// TIA Portal V19 export
FUNCTION "A0301_Fermi_P3_CALL" : Void   // FC120, LAD
// stored: SetENOAutomatically false
BEGIN

REGION Network 1 (SCL): << TRASFERIMENTO stati CIn del blocco >>
   // TRASFERIMENTO #CIn MANAGER
   "A0301_Fermi_P3".CIn.Manager := "A0301_Manager".COut.P3.Fermi;
   //
   "A0301_Fermi_P3".CIn.SemiAut := "A0301_Manager".DataIn.SemiAut_Pb;

   // Trasferimento status alla Stazione P2 da COut a Cin delle stazioni successive
   "A0301_Fermi_P3".CIn.P2.Fermi := "A0301_Fermi_P2".COut.Fermi;

   // Trasferimento status alla Stazione P3 da COut a Cin del sollevatore P2
   "A0301_Fermi_P3".CIn.P2.Sollevatore := "A0301_Fermi_P2".COut.Sollevatori;

   // Trasferimenti status lettura posizioni Trasporto al Cin delle stazioni
   "A0301_Fermi_P3".CIn.Trasporto := "A0301_Trasporto".COut.Ax;
END_REGION

REGION Network 2 (SCL): << TRASFERIMENTO stati DataIn >>
   // SOSTITUIRE SYS.BAYPASS
   // TRASFERIMENTO #DataIn STATI BUTTON STAZIONE P3

   REGION TRASFERIMENTO DataIn DIGITAL INPUT dei LIMIT SWITCH

       // Trasferimento ingressi digitali Limit Switch Fermi P3
       // 
       "A0301_Fermi_P3".Fermi[1].DataIn.Rest_Ls[1] := "A0301_CinghiaTrasporto_1.2_Ls_Rest_1";
       "A0301_Fermi_P3".Fermi[2].DataIn.Rest_Ls[1] := "A0301_CinghiaTrasporto_2.2_Ls_Rest_1";
       "A0301_Fermi_P3".Fermi[3].DataIn.Rest_Ls[1] := "A0301_CinghiaTrasporto_3.2_Ls_Rest_1";
       "A0301_Fermi_P3".Fermi[4].DataIn.Rest_Ls[1] := "A0301_CinghiaTrasporto_4.2_Ls_Rest_1";
       "A0301_Fermi_P3".Fermi[5].DataIn.Rest_Ls[1] := "A0301_CinghiaTrasporto_5.2_Ls_Rest_1";
       "A0301_Fermi_P3".Fermi[6].DataIn.Rest_Ls[1] := "A0301_CinghiaTrasporto_6.2_Ls_Rest_1";

   END_REGION ;
END_REGION

REGION Network 3: DataIn - Fermi
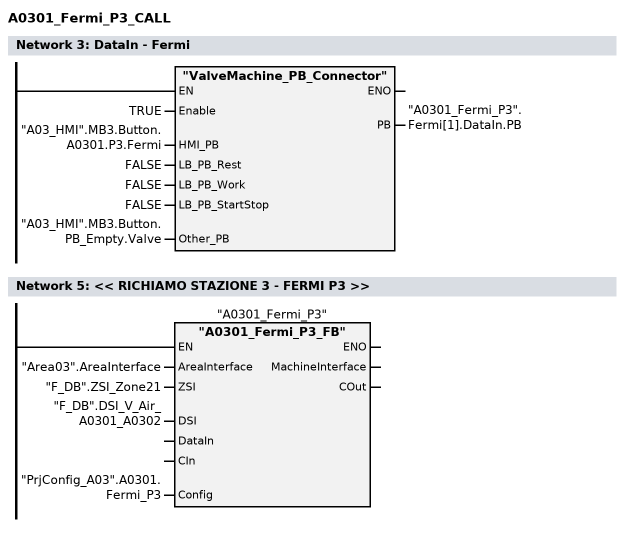
   RUNG wire#powerrail
      "ValveMachine_PB_Connector"(Enable := TRUE, HMI_PB := "A03_HMI".MB3.Button.A0301.P3.Fermi, LB_PB_Rest := FALSE, LB_PB_Work := FALSE, LB_PB_StartStop := FALSE, Other_PB := "A03_HMI".MB3.Button.PB_Empty.Valve, PB => "A0301_Fermi_P3".Fermi[1].DataIn.PB)
   END_RUNG
   // the same network as SCL:
   "ValveMachine_PB_Connector"(Enable := TRUE,
                           HMI_PB := "A03_HMI".MB3.Button.A0301.P3.Fermi,
                           LB_PB_Rest := FALSE,
                           LB_PB_Work := FALSE,
                           LB_PB_StartStop := FALSE,
                           Other_PB := "A03_HMI".MB3.Button.PB_Empty.Valve,
                           PB => "A0301_Fermi_P3".Fermi[1].DataIn.PB);
END_REGION

REGION Network 4 (SCL): DataIn - Fermi [1..6]
   // TRASFERIMENTO STATO PULSANTI - Comando manuale diretto 
   "A0301_Fermi_P3".Fermi[6].DataIn.PB.Rest := "A0301_Fermi_P3".Fermi[5].DataIn.PB.Rest := "A0301_Fermi_P3".Fermi[4].DataIn.PB.Rest :=
   "A0301_Fermi_P3".Fermi[3].DataIn.PB.Rest := "A0301_Fermi_P3".Fermi[2].DataIn.PB.Rest := "A0301_Fermi_P3".Fermi[1].DataIn.PB.Rest;

   "A0301_Fermi_P3".Fermi[6].DataIn.PB.Work := "A0301_Fermi_P3".Fermi[5].DataIn.PB.Work := "A0301_Fermi_P3".Fermi[4].DataIn.PB.Work :=
   "A0301_Fermi_P3".Fermi[3].DataIn.PB.Work := "A0301_Fermi_P3".Fermi[2].DataIn.PB.Work := "A0301_Fermi_P3".Fermi[1].DataIn.PB.Work;
END_REGION

REGION Network 5: << RICHIAMO STAZIONE 3 - FERMI P3 >>
   RUNG wire#powerrail
      "A0301_Fermi_P3"(AreaInterface := "Area03".AreaInterface, ZSI := "F_DB".ZSI_Zone21, DSI := "F_DB".DSI_V_Air_A0301_A0302, DataIn :=, CIn :=, Config := "PrjConfig_A03".A0301.Fermi_P3, MachineInterface =>, COut =>)
   END_RUNG
   // the same network as SCL:
   "A0301_Fermi_P3"(AreaInterface := "Area03".AreaInterface,   // "A0301_Fermi_P3_FB"
                    ZSI := "F_DB".ZSI_Zone21,
                    DSI := "F_DB".DSI_V_Air_A0301_A0302,
                    Config := "PrjConfig_A03".A0301.Fermi_P3);
END_REGION

REGION Network 6 (SCL): << TRASFERIMENTO stati DataOut >>
    REGION COMANDO DELLE USCITE FERMI P3

       // Fermi blocco prodotto Stazione P3 - RIPOSO

        "A0301_CinghiaTrasporto_1.2_V_Rest_1" := "A0301_Fermi_P3".Fermi[1].DataOut.RestSolenoid;
        "A0301_CinghiaTrasporto_2.2_V_Rest_1" := "A0301_Fermi_P3".Fermi[2].DataOut.RestSolenoid;
        "A0301_CinghiaTrasporto_3.2_V_Rest_1" := "A0301_Fermi_P3".Fermi[3].DataOut.RestSolenoid;
        "A0301_CinghiaTrasporto_4.2_V_Rest_1" := "A0301_Fermi_P3".Fermi[4].DataOut.RestSolenoid;
        "A0301_CinghiaTrasporto_5.2_V_Rest_1" := "A0301_Fermi_P3".Fermi[5].DataOut.RestSolenoid;
        "A0301_CinghiaTrasporto_6.2_V_Rest_1" := "A0301_Fermi_P3".Fermi[6].DataOut.RestSolenoid;

       // Fermi blocco prodotto Stazione P3 - LAVORO
       // 
        "A0301_CinghiaTrasporto_1.2_V_Work_2" := "A0301_Fermi_P3".Fermi[1].DataOut.WorkSolenoid;
        "A0301_CinghiaTrasporto_2.2_V_Work_2" := "A0301_Fermi_P3".Fermi[2].DataOut.WorkSolenoid;
        "A0301_CinghiaTrasporto_3.2_V_Work_2" := "A0301_Fermi_P3".Fermi[3].DataOut.WorkSolenoid;
        "A0301_CinghiaTrasporto_4.2_V_Work_2" := "A0301_Fermi_P3".Fermi[4].DataOut.WorkSolenoid;
        "A0301_CinghiaTrasporto_5.2_V_Work_2" := "A0301_Fermi_P3".Fermi[5].DataOut.WorkSolenoid;
        "A0301_CinghiaTrasporto_6.2_V_Work_2" := "A0301_Fermi_P3".Fermi[6].DataOut.WorkSolenoid;

   END_REGION ;
END_REGION
END_FUNCTION
